KUKA KRL program: mnt_after_brl_find.src, mnt_after_brl_find.dat

--- mnt_after_brl_find.src ---
&ACCESS RVO1
&REL 4
&PARAM DISKPATH = KRC:\R1\Program\Production
DEF mnt_after_brl_find( )
   ;FOLD INI;%{PE}
      ;FOLD BASISTECH INI
         GLOBAL INTERRUPT DECL 3 WHEN $STOPMESS==TRUE DO IR_STOPM ( )
         INTERRUPT ON 3
         BAS (#INITMOV,0 )
      ;ENDFOLD (BASISTECH INI)
      ;FOLD USER INI
         ;Make your modifications here

      ;ENDFOLD (USER INI)
   ;ENDFOLD (INI)

   Xdummy_point = $POS_ACT
   PTP Xdummy_point
   homepos()

   ;FOLD HandShake[5 : At Maintenance Position], WAIT on Response
;FOLD ;%{h}
;Params IlfProvider=model3_handshakectrl; Core_CmdTechHandShake=HandShake; Core_CmdHandShake=5; Core_Wait=True
;ENDFOLD
HandShake_Set (5,false)
HandShake_Check (5,false)
;ENDFOLD



PTP Xdummy_point
   ;FOLD HandShake[24 : Maintenance Done Returned to Barrel], WAIT on Response
;FOLD ;%{h}
;Params IlfProvider=model3_handshakectrl; Core_CmdTechHandShake=HandShake; Core_CmdHandShake=24; Core_Wait=True
;ENDFOLD
HandShake_Set (24,false)
HandShake_Check (24,false)
;ENDFOLD

   Exit_Program()


END

--- mnt_after_brl_find.dat ---
&ACCESS RVO1
&REL 4
&PARAM DISKPATH = KRC:\R1\Program\Production
DEFDAT  mnt_after_brl_find
;FOLD EXTERNAL DECLARATIONS;%{PE}%MKUKATPBASIS,%CEXT,%VCOMMON,%P
;FOLD BASISTECH EXT;%{PE}%MKUKATPBASIS,%CEXT,%VEXT,%P
EXT  BAS (BAS_COMMAND  :IN,REAL  :IN )
DECL INT SUCCESS
;ENDFOLD (BASISTECH EXT)
;FOLD USER EXT;%{E}%MKUKATPUSER,%CEXT,%VEXT,%P
;Make your modifications here

;ENDFOLD (USER EXT)
;ENDFOLD (EXTERNAL DECLARATIONS)
DECL E6POS Xweld_pos={X -85.9545,Y -1068.13318,Z 1203.34253,A 9.17978477,B 0.595385969,C 45.0561867,S 6,T 18,E1 0.0,E2 0.0,E3 0.0,E4 0.0,E5 0.0,E6 0.0}
DECL FDAT Fweld_pos={TOOL_NO 1,BASE_NO 0,IPO_FRAME #BASE,POINT2[] " "}
DECL MODULEPARAM_T LAST_TP_PARAMS={PARAMS[] "Kuka.VelocityFieldEnabled=True; Kuka.ColDetectFieldEnabled=True; Kuka.MovementParameterFieldEnabled=True; Kuka.IsAngleEnabled=False; Kuka.PointName=weld_pos; Kuka.FrameData.base_no=0; Kuka.FrameData.tool_no=1; Kuka.FrameData.ipo_frame=#BASE; Kuka.FrameData.point2=; Kuka.isglobalpoint=False; Kuka.VelocityPtp=5; Kuka.BlendingEnabled=False; Kuka.CurrentCDSetIndex=0   "}
DECL FDAT FHOME2={TOOL_NO 1,BASE_NO 0,IPO_FRAME #BASE,POINT2[] " "}
DECL BASIS_SUGG_T LAST_BASIS={POINT1[] "home7                   ",POINT2[] "home7                   ",CP_PARAMS[] "CPDAT0                  ",PTP_PARAMS[] "PDAT4                   ",CONT[] "                        ",CP_VEL[] "2.0                     ",PTP_VEL[] "30                      ",SYNC_PARAMS[] "SYNCDAT                 ",SPL_NAME[] "S0                      ",A_PARAMS[] "ADAT0                   "}
DECL FDAT Fhome4={TOOL_NO 1,BASE_NO 0,IPO_FRAME #BASE,POINT2[] " ",TQ_STATE FALSE}
DECL PDAT PPDAT1={VEL 100.000,ACC 5.00000,APO_DIST 100.000,APO_MODE #CDIS,GEAR_JERK 50.0000,EXAX_IGN 0}
DECL FDAT Fhome3={TOOL_NO 1,BASE_NO 0,IPO_FRAME #BASE,POINT2[] " ",TQ_STATE FALSE}
DECL PDAT PPDAT2={VEL 100.000,ACC 5.00000,APO_DIST 100.000,APO_MODE #CDIS,GEAR_JERK 50.0000,EXAX_IGN 0}
DECL E6POS XHOME6={X 403.077454,Y 1348.19373,Z 1142.98474,A -164.725662,B -89.6085281,C 100.191284,S 6,T 51,E1 0.0,E2 0.0,E3 0.0,E4 0.0,E5 0.0,E6 0.0}
DECL FDAT Fhome6={TOOL_NO 1,BASE_NO 0,IPO_FRAME #BASE,POINT2[] " ",TQ_STATE FALSE}
DECL PDAT PPDAT3={VEL 100.000,ACC 5.00000,APO_DIST 100.000,APO_MODE #CDIS,GEAR_JERK 50.0000,EXAX_IGN 0}
DECL E6POS XHOME7={X 403.077454,Y 1348.19373,Z 1142.98474,A -164.725662,B -89.6085281,C 100.191284,S 6,T 51,E1 0.0,E2 0.0,E3 0.0,E4 0.0,E5 0.0,E6 0.0}
DECL FDAT Fhome7={TOOL_NO 1,BASE_NO 0,IPO_FRAME #BASE,POINT2[] " ",TQ_STATE FALSE}
DECL PDAT PPDAT4={VEL 100.000,ACC 5.00000,APO_DIST 100.000,APO_MODE #CDIS,GEAR_JERK 50.0000,EXAX_IGN 0}
ENDDAT
